(* PLC project Desconhecido, Desconhecido Sem nome 1 *)
(* stored: creationDateTime 1970-01-01T12:13:12, modificationDateTime 1970-01-01T12:14:12 *)

PROGRAM instance0

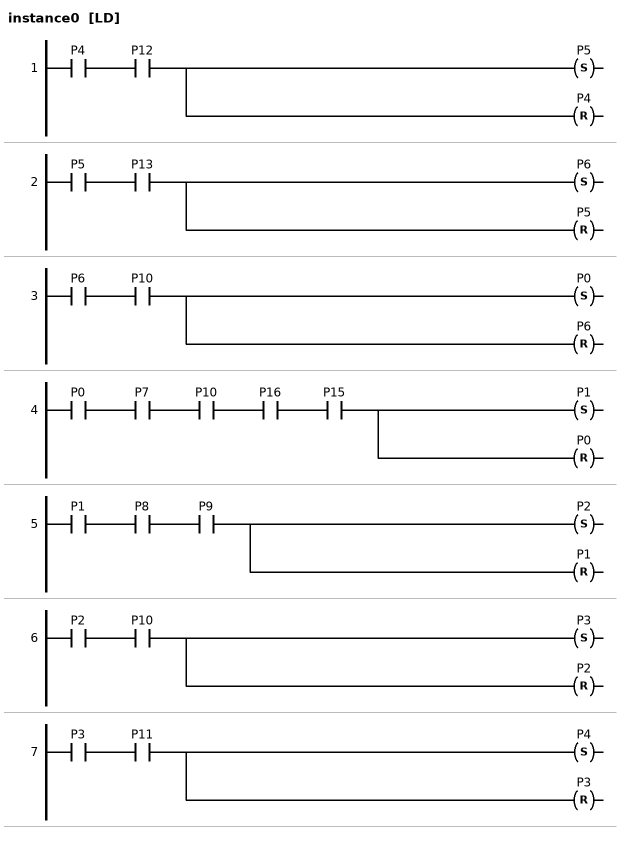
(* LD diagram, written out as Structured Text *)
IF P4 AND P12 THEN P5 := TRUE; END_IF;
IF P4 AND P12 THEN P4 := FALSE; END_IF;
IF P5 AND P13 THEN P6 := TRUE; END_IF;
IF P5 AND P13 THEN P5 := FALSE; END_IF;
IF P6 AND P10 THEN P0 := TRUE; END_IF;
IF P6 AND P10 THEN P6 := FALSE; END_IF;
IF P0 AND P7 AND P10 AND P16 AND P15 THEN P1 := TRUE; END_IF;
IF P0 AND P7 AND P10 AND P16 AND P15 THEN P0 := FALSE; END_IF;
IF P1 AND P8 AND P9 THEN P2 := TRUE; END_IF;
IF P1 AND P8 AND P9 THEN P1 := FALSE; END_IF;
IF P2 AND P10 THEN P3 := TRUE; END_IF;
IF P2 AND P10 THEN P2 := FALSE; END_IF;
IF P3 AND P11 THEN P4 := TRUE; END_IF;
IF P3 AND P11 THEN P3 := FALSE; END_IF;
END_PROGRAM

CONFIGURATION config0
  RESOURCE resource1 ON PLC
    TASK task0(INTERVAL := T#20ms, PRIORITY := 0);
    PROGRAM instance0 WITH task0 : program0;
  END_RESOURCE
END_CONFIGURATION
